// TIA Portal V20 export
// export: Created 2025-12-01T14:57:05.5491465Z, ExportSetting None, DisplayName Totally Integrated Automation Portal, DisplayVersion V20 Update 3, DisplayName TIA Portal Openness, DisplayVersion V20 Update 3, DisplayName TIA Portal Version Control Interface, DisplayVersion V20 Update 3, DisplayName STEP 7 Professional, DisplayVersion V20 Update 3, DisplayName STEP 7 Safety, DisplayVersion V20 Update 2, DisplayName WinCC Basic/Comfort/Advanced, DisplayVersion V20 Update 3, DisplayName WinCC Professional, DisplayVersion V20 Update 3, DisplayName WinCC Unified, DisplayVersion V20 Update 3
FUNCTION "FC892_Obtener_ValorDelAtributo" : Void   // FC892, LAD
TITLE = "ObtemerValorAtributo" - Convertir a Doble Entero una String
{ S7_Optimized_Access := 'FALSE' }
AUTHOR : TRACKING
NAME : 20130301
VERSION : 3.0
// stored: AutoNumber false, SetENOAutomatically false
   VAR_INPUT
      DB_String : Word;   // DB donde esta la String
      OffsetIni : UInt;   // Numero de byte de la String donde empieza
   END_VAR
   VAR_OUTPUT
      Valor : UDInt;   // Valor de la Conversion
   END_VAR
   VAR_TEMP
      PunteroDB : DWord;   // Puntero al DB de la String
      NumDB : Word;   // Numero de DB de la String
      OffsetActual : UInt;   // Numero de bytes de la String Actual
      TEMP_Valor : UDInt;
   END_VAR
BEGIN

NETWORK
TITLE = Inicializaciones
// Inicializar las Variables que se necesitan
      L     0;  // Inicializo el Valor a 0 (TEMPORAL)
      T     #TEMP_Valor;

      L     #DB_String;
      T     #NumDB;

      L     #OffsetIni;  // Apunta al primer caracter el de Mayor peso
      T     #OffsetActual;

NETWORK
TITLE = Cuerpo de la Funcion
// - Calcula el Puntero al Caracter a Convertir
// - Se mira si es Numero
// - Obteniendo el Nuevo Valor de la Conversion
// - Pasar al siguiente Caracter
// ----------------------------------------------------------------------------------------
// Calcula el Puntero al Caracter a Convertir

InicioBucle:OPN   DB [#NumDB];
      L     #OffsetActual;
      SLD   3;
      T     #PunteroDB;

// ----------------------------------------------------------------------------------------
// Se mira si es numero

      L     DBB [#PunteroDB];
      L     '0';
      <I;
      JC    Final;
      L     DBB [#PunteroDB];
      L     '9';
      >I;
      JC    Final;

// ----------------------------------------------------------------------------------------
// Obteniendo el Nuevo Valor de la Conversion

      L     #TEMP_Valor;  // Un digito más para el Valor
      L     10;  // Mutiplico por 10
      *D;
      T     #TEMP_Valor;

      L     DBB [#PunteroDB];  // Quito la parte Alta del Byte Leido
      L     W#16#F;  // Es como restar w#16#30
      AD;
      L     #TEMP_Valor;  // Y lo sumo
      +D;
      T     #TEMP_Valor;


// ----------------------------------------------------------------------------------------
// Pasar al siguiente caracter

      L     #OffsetActual;  // Continuo para ver si el siguiente es digito
      L     1;
      +I;
      T     #OffsetActual;
      JU    InicioBucle;



NETWORK
TITLE = Final
// Final de la Funcion
Final:NOP   0;

      L     #TEMP_Valor;  // Activo la Salida
      T     #Valor;



END_FUNCTION
